FUNCTION_BLOCK FINAL OnRequestError EXTENDS AwaitableError

END_FUNCTION_BLOCK

(* stored: Version 1.1.0.1, ProductVersion 3.1.4024.12
   POU OnRequestError: Id {3196f5e9-f6dc-4fe4-8eda-29b243c11ef9}, SpecialFunc None *)
